// TIA Portal V20 export
FUNCTION "V101" : Void   // FC17, FBD
{ S7_Optimized_Access := 'TRUE' }
// stored: SetENOAutomatically false
   VAR_TEMP
      Temp : "DigVal";
      Temp_1 : "DigVal";
      State : "Service_States";
   END_VAR
BEGIN

REGION Network 1: Channel input
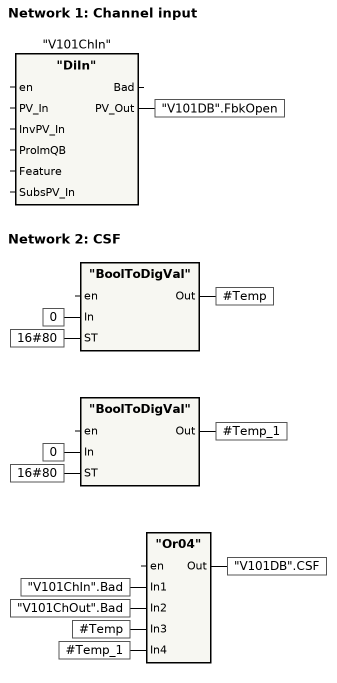
   "V101ChIn"(PV_Out => "V101DB".FbkOpen);   // "DiIn"
END_REGION

REGION Network 2: CSF
   "BoolToDigVal"(In := 0, ST := 16#80, Out => #Temp);
   "BoolToDigVal"(In := 0, ST := 16#80, Out => #Temp_1);
   "Or04"(In1 := "V101ChIn".Bad, In2 := "V101ChOut".Bad, In3 := #Temp, In4 := #Temp_1, Out => "V101DB".CSF);
END_REGION

REGION Network 3: VlvAn Intlock
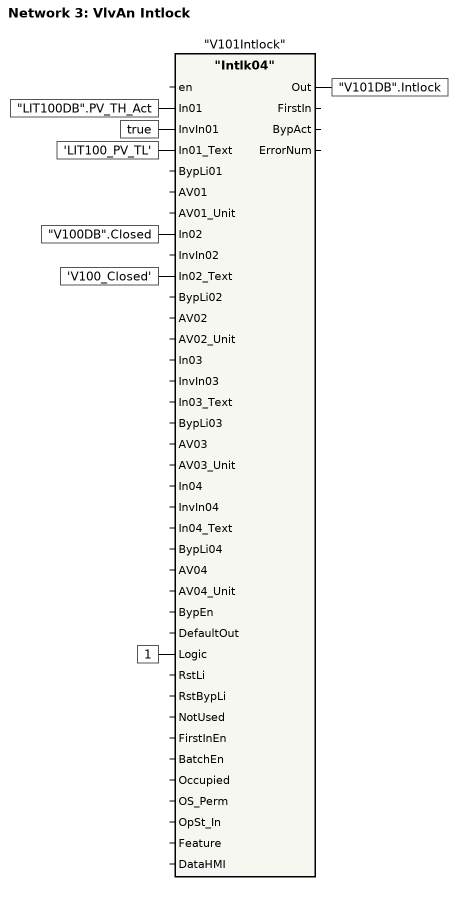
   "V101Intlock"(In01 := "LIT100DB".PV_TH_Act,   // "Intlk04"
                 InvIn01 := true,
                 In01_Text := 'LIT100_PV_TL',
                 In02 := "V100DB".Closed,
                 In02_Text := 'V100_Closed',
                 Logic := 1,
                 Out => "V101DB".Intlock);
END_REGION

REGION Network 4: VlvAnL
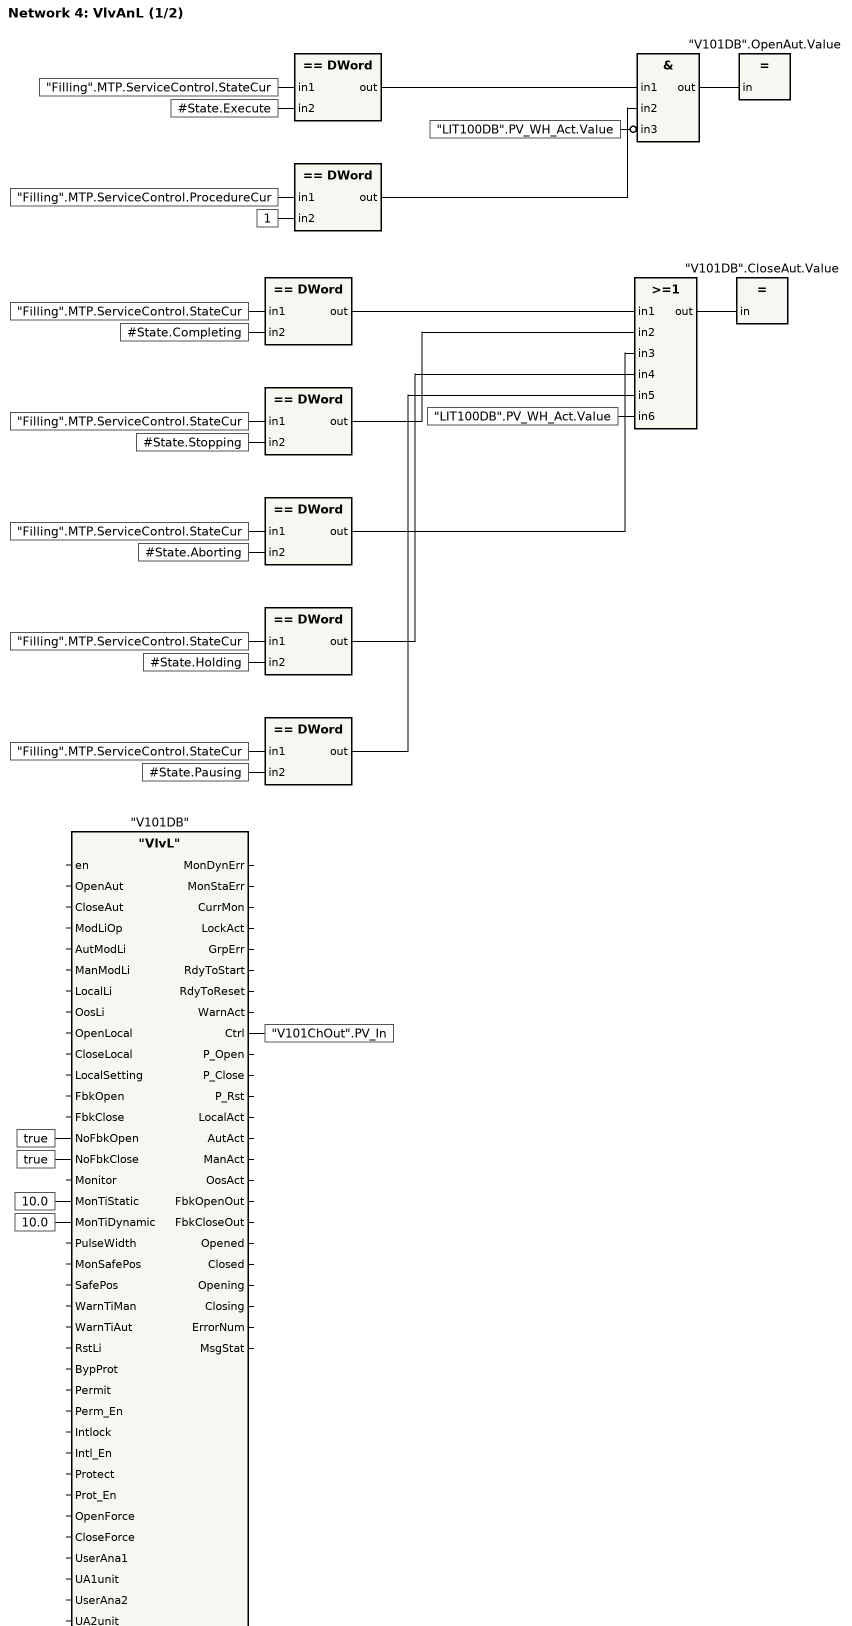
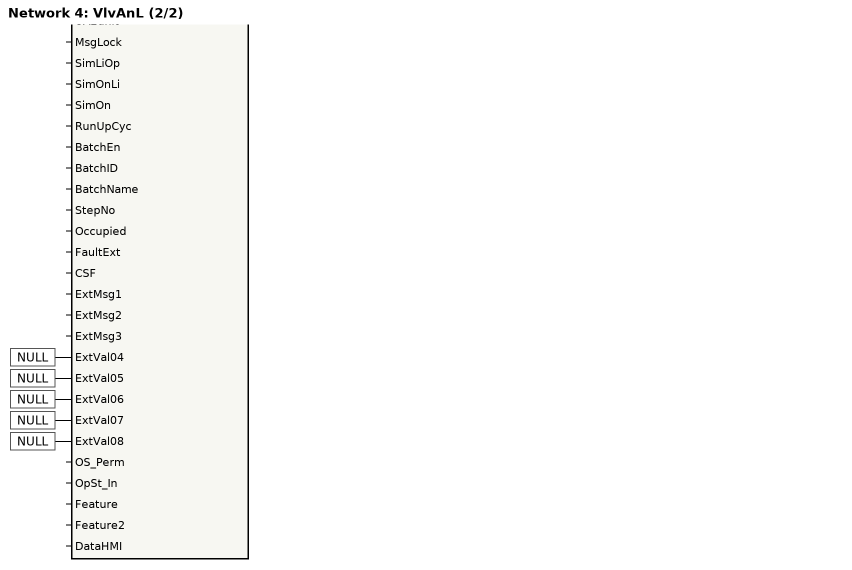
   "V101DB".OpenAut.Value := ("Filling".MTP.ServiceControl.StateCur = #State.Execute) AND ("Filling".MTP.ServiceControl.ProcedureCur = 1) AND NOT "LIT100DB".PV_WH_Act.Value;
   "V101DB".CloseAut.Value := ("Filling".MTP.ServiceControl.StateCur = #State.Completing) OR ("Filling".MTP.ServiceControl.StateCur = #State.Stopping) OR ("Filling".MTP.ServiceControl.StateCur = #State.Aborting) OR ("Filling".MTP.ServiceControl.StateCur = #State.Holding) OR ("Filling".MTP.ServiceControl.StateCur = #State.Pausing) OR "LIT100DB".PV_WH_Act.Value;
   "V101DB"(NoFbkOpen := true,   // "VlvL"
            NoFbkClose := true,
            MonTiStatic := 10.0,
            MonTiDynamic := 10.0,
            ExtVal04 := NULL,
            ExtVal05 := NULL,
            ExtVal06 := NULL,
            ExtVal07 := NULL,
            ExtVal08 := NULL,
            Ctrl => "V101ChOut".PV_In);
END_REGION

REGION Network 5: MTP
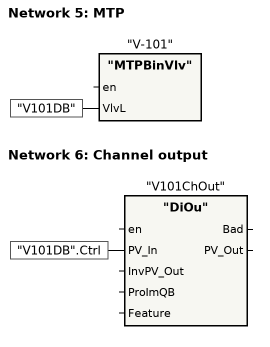
   "V-101"(VlvL := "V101DB");   // "MTPBinVlv"
END_REGION

REGION Network 6: Channel output
   "V101ChOut"(PV_In := "V101DB".Ctrl);   // "DiOu"
END_REGION
END_FUNCTION
